FUNCTION_BLOCK FB_RobotInterefaceMAIN
VAR_INPUT
	bEnable :BOOL; // PLC Logic Enable
	bInputConvReady :BOOL; // Signal from input conveyor: box is ready at robot pickup position
	bOutputConvReady :BOOL; // Signal from output conveyor: drop zone is clear
	
END_VAR

VAR_OUTPUT
	bRobotReadyPickInputConv :BOOL; // Permission to robot: OK to pick from input conveyor
	bRobotReadyPlaceOutputConv :BOOL; // Permission to robot: OK to place on output conveyor
	
END_VAR
VAR
	
END_VAR

IF bEnable THEN
	bRobotReadyPickInputConv := TRUE;
	bRobotReadyPlaceOutputConv := TRUE;
ELSE
	bRobotReadyPickInputConv := FALSE;
	bRobotReadyPlaceOutputConv := FALSE;
END_IF

END_FUNCTION_BLOCK

(* stored: Version 1.1.0.1, ProductVersion 3.1.4026.17
   POU FB_RobotInterefaceMAIN: Id {57ef01b0-8444-4a14-b048-721777179cc2}, SpecialFunc None *)
